{attribute 'GeneratedUsingTerminal: AT2050-0500-0023'}
{attribute addProperty BoxType "AT2050-0500-0023"}
{attribute addProperty Id "A_0090_AT2050_5501_0019_AT2050_5501AT2050_33A3DF1B80"}
{attribute addProperty CRC "3002261333"}
{attribute addProperty Size "80"}
TYPE A_0054_AT2050_0500_0023_B2F2DF55 EXTENDS AT2050_A7FEA1CF :
STRUCT
	{attribute addProperty Name "A_0090_AT2050_5501_0019_AT2050_5501"}
	{attribute addProperty PreviousPort "A_0054(AT2050-0500-0023) : B"}
	A_0090_AT2050_5501_0019_AT2050_5501 : AT2050_33A3DF1B;
END_STRUCT
END_TYPE

(* stored: Version 1.2.0.0, ProductVersion 3.1.4024.9
   DUT A_0054_AT2050_0500_0023_B2F2DF55: Id {fccf94b5-e00f-472b-b21b-83e9272b9c98} *)
